// TwinCAT 3 PLC project SZ2_Library
// ProgramVersion: 3.1.4024.0
// libraries:
//   Tc2_Standard, * (Beckhoff Automation GmbH)
//   Tc2_System, * (Beckhoff Automation GmbH)
//   Tc3_Module, * (Beckhoff Automation GmbH)
// project tree:
//   / PlcTask.TcTTO
//   POUs/Function Blocks/ FB_HeatingLoop.TcPOU, FB_PID_Simulation.TcPOU, FB_Simu_NT.TcPOU
//   POUs/Functions/ fcWriteOutput.TcPOU
//   POUs/ MAIN.TcPOU
// real-time tasks:
//   TASK PlcTask: cycle T#10ms, priority 20, ADS port 350

CONFIGURATION SZ2_Library
    RESOURCE PLC ON TwinCAT3
        TASK PlcTask(INTERVAL := T#10ms, PRIORITY := 20);
        PROGRAM MAIN WITH PlcTask : MAIN;
    END_RESOURCE
END_CONFIGURATION

// ---- POUs/MAIN.TcPOU
PROGRAM MAIN
VAR
	FB_Test1		: FB_HeatingLoop;
	
	rPID_Core		: REAL;
	rPID_SUrface	: REAL;
	abIN_HE_Fault	: ARRAY [1..12] OF BOOL;
	
	iT_Core			: INT;
	iT_Surface		: INT;
	rmA				: REAL;
	bCore_Fault		: BOOL;
	bSurface_Fault	: BOOL;
	abOUT_HE_Fault	: ARRAY [1..12] OF BOOL;
END_VAR

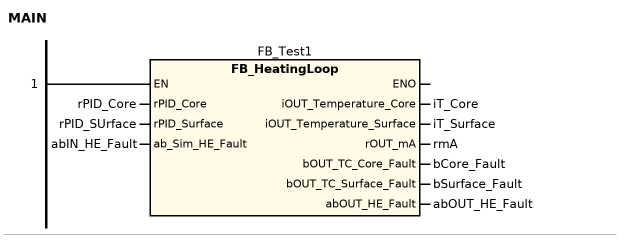
// NETWORK 1
FB_Test1(
    rPID_Core := rPID_Core,
    rPID_Surface := rPID_SUrface,
    ab_Sim_HE_Fault := abIN_HE_Fault,
    iOUT_Temperature_Core => iT_Core,
    iOUT_Temperature_Surface => iT_Surface,
    rOUT_mA => rmA,
    bOUT_TC_Core_Fault => bCore_Fault,
    bOUT_TC_Surface_Fault => bSurface_Fault,
    abOUT_HE_Fault => abOUT_HE_Fault); // FB_HeatingLoop

END_PROGRAM

// ---- POUs/Function Blocks/FB_HeatingLoop.TcPOU
FUNCTION_BLOCK FB_HeatingLoop
VAR_INPUT
	rPID_Core				: REAL;
	rPID_Surface			: REAL;
	ab_Sim_HE_Fault			: ARRAY [1..12] OF BOOL;
END_VAR
VAR_OUTPUT
	iOUT_Temperature_Core		: INT;
	iOUT_Temperature_Surface	: INT;
	rOUT_mA						: REAL;
	bOUT_TC_Core_Fault			: BOOL;
	bOUT_TC_Surface_Fault		: BOOL;	
	abOUT_HE_Fault				: ARRAY [1..12] OF BOOL;
END_VAR

VAR
	FB_Sim_Core_1			: FB_PID_Simulation;
	FB_Sim_Core_2			: FB_PID_Simulation;
	FB_Sim_Surface_1		: FB_PID_Simulation;
	FB_Sim_Surface_2		: FB_PID_Simulation;
	
	rTemperature_Core		: REAL;
	rTemperatrue_Surface	: REAL;
	
// Temp Variables
	rTempC				: REAL;
	rTempC_2			: REAL;
	rPID_Core_Temp		: REAL;
	rTempS				: REAL;
	rTempS_2			: REAL;

END_VAR
VAR // added by the converter: edge detectors and wires of the graphical bodies
    _w1 : BOOL;
END_VAR

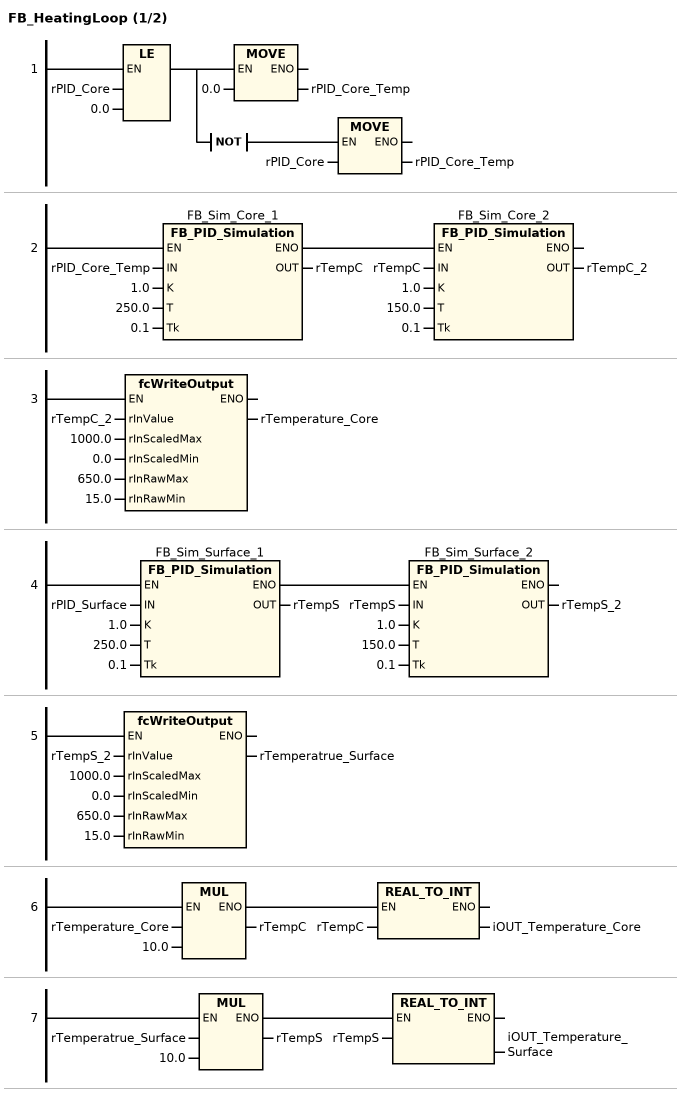
// NETWORK 1
_w1 := rPID_Core <= 0.0;
IF _w1 THEN rPID_Core_Temp := 0.0; END_IF
IF NOT _w1 THEN rPID_Core_Temp := rPID_Core; END_IF

// NETWORK 2
FB_Sim_Core_1(IN := rPID_Core_Temp, K := 1.0, T := 250.0, Tk := 0.1, OUT => rTempC); // FB_PID_Simulation
FB_Sim_Core_2(IN := rTempC, K := 1.0, T := 150.0, Tk := 0.1, OUT => rTempC_2); // FB_PID_Simulation

// NETWORK 3
rTemperature_Core := fcWriteOutput(rInValue := rTempC_2, rInScaledMax := 1000.0, rInScaledMin := 0.0, rInRawMax := 650.0, rInRawMin := 15.0);

// NETWORK 4
FB_Sim_Surface_1(IN := rPID_Surface, K := 1.0, T := 250.0, Tk := 0.1, OUT => rTempS); // FB_PID_Simulation
FB_Sim_Surface_2(IN := rTempS, K := 1.0, T := 150.0, Tk := 0.1, OUT => rTempS_2); // FB_PID_Simulation

// NETWORK 5
rTemperatrue_Surface := fcWriteOutput(rInValue := rTempS_2, rInScaledMax := 1000.0, rInScaledMin := 0.0, rInRawMax := 650.0, rInRawMin := 15.0);

// NETWORK 6
rTempC := rTemperature_Core * 10.0;
iOUT_Temperature_Core := REAL_TO_INT(rTempC);

// NETWORK 7
rTempS := rTemperatrue_Surface * 10.0;
iOUT_Temperature_Surface := REAL_TO_INT(rTempS);

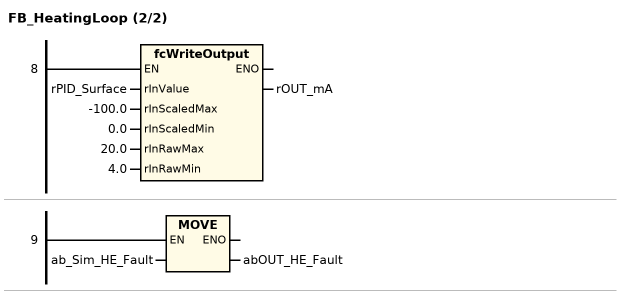
// NETWORK 8
rOUT_mA := fcWriteOutput(rInValue := rPID_Surface, rInScaledMax := -100.0, rInScaledMin := 0.0, rInRawMax := 20.0, rInRawMin := 4.0);

// NETWORK 9
abOUT_HE_Fault := ab_Sim_HE_Fault;

END_FUNCTION_BLOCK

// ---- POUs/Function Blocks/FB_PID_Simulation.TcPOU
FUNCTION_BLOCK FB_PID_Simulation
VAR_INPUT
	IN		: REAL;
	K		: REAL;
	T		: REAL;
	Tk		: REAL;
END_VAR
VAR_OUTPUT
	OUT		: REAL;
END_VAR
VAR
END_VAR

OUT	:=	(Tk*K*IN+T*OUT)/(T+Tk);

END_FUNCTION_BLOCK

// ---- POUs/Functions/fcWriteOutput.TcPOU
FUNCTION fcWriteOutput : REAL
//Writes a scaled output

VAR_INPUT
	rInValue	: REAL;		// Input value
	rInScaledMax	: REAL;		// Engineering units range max
	rInScaledMin	: REAL;		// Engineering units range min
	rInRawMax		: REAL;		// Raw maximum - overflow limit
	rInRawMin		: REAL;		// Raw minimum - underflow limit
END_VAR
VAR
	rTemp			: REAL;		// Temp REAL value
	rRawMax			: REAL;
	rRawMin			: REAL;
	rRawRange		: REAL;
	rScaledRange	: REAL;
	rOutput			: REAL;
	iOutput			: INT;
END_VAR

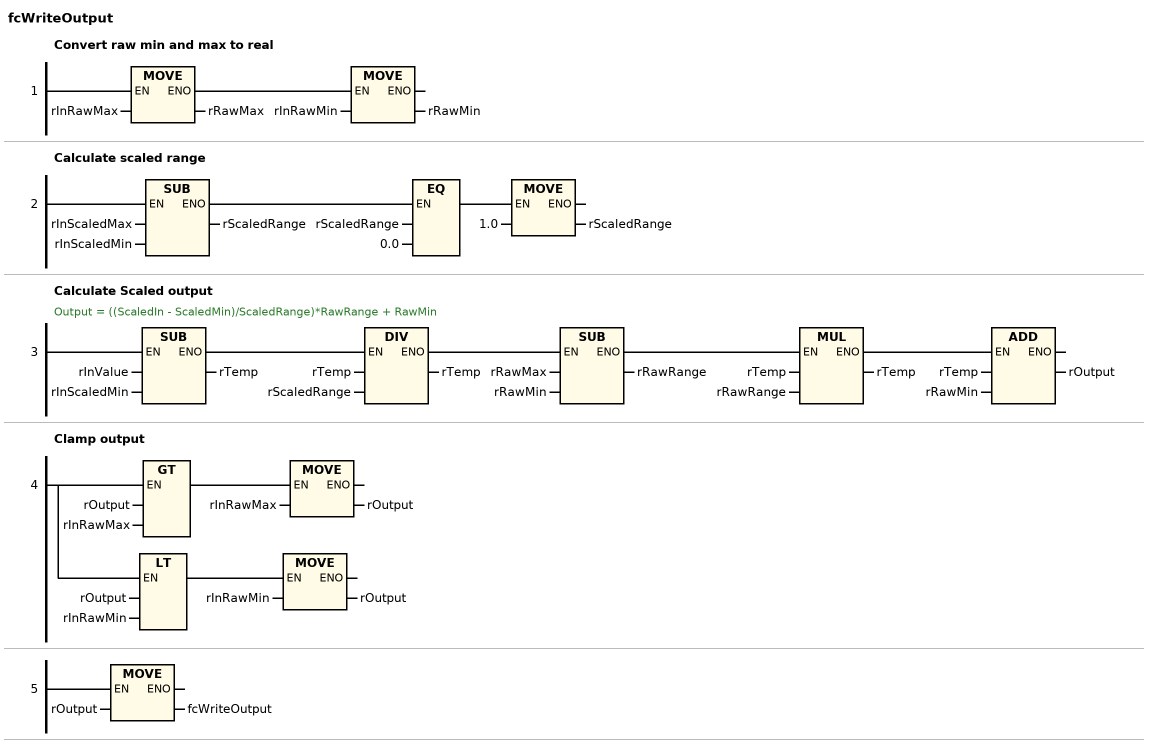
// NETWORK 1: Convert raw min and max to real
rRawMax := rInRawMax;
rRawMin := rInRawMin;

// NETWORK 2: Calculate scaled range
rScaledRange := rInScaledMax - rInScaledMin;
IF rScaledRange = 0.0 THEN rScaledRange := 1.0; END_IF

// NETWORK 3: Calculate Scaled output
// Output = ((ScaledIn - ScaledMin)/ScaledRange)*RawRange + RawMin
rTemp := rInValue - rInScaledMin;
rTemp := rTemp / rScaledRange;
rRawRange := rRawMax - rRawMin;
rTemp := rTemp * rRawRange;
rOutput := rTemp + rRawMin;

// NETWORK 4: Clamp output
IF rOutput > rInRawMax THEN rOutput := rInRawMax; END_IF
IF rOutput < rInRawMin THEN rOutput := rInRawMin; END_IF

// NETWORK 5
fcWriteOutput := rOutput;

END_FUNCTION

// ---- POUs/Function Blocks/FB_Simu_NT.TcPOU
FUNCTION_BLOCK FB_Simu_NT
VAR_INPUT

END_VAR

VAR_OUTPUT
	iOUT_TC_Water_1			: INT;
	iOUT_TC_Water_2			: INT;
	iOUT_CJC_Value			: INT;
	iOUT_ToolID_Value		: INT;
	bOUT_WaterFlow_1		: BOOL;
	bOUT_WaterFlow_2		: BOOL;
	bOUT_AirPressure		: BOOL;
	bOUT_TC_Water_1_Error	: BOOL;
	bOUT_TC_Water_2_Error	: BOOL;
	bOUT_CJC_Error			: BOOL;
	bOUT_ToolID_Error		: INT;
END_VAR
VAR
END_VAR

// NETWORK 1

END_FUNCTION_BLOCK
